// TIA Portal V18 export
TYPE "PLCtoMES_MainCheckOut"
// stored: IsFailsafeCompliant false
   STRUCT
      "P-DataSaveReq" : Bool;   // PLC请求采集质量数据标志位（质量数据全部刷新后触发）MES置位M-DataDone采集完成标志位后，由PLC复位此信号。
      "P-PartType" : String[28];   // PLC请求MES保存时发送产品型号（有RFID则从RFID读取，无RFID，从扫码枪获取）
      "P-PartID" : Array[1..10] of String[48];   // PLC请求MES保存时发送产品序列号（有RFID则从RFID读取，无RFID，从扫码枪获取）
      "P-SubPartID" : Array[1..10] of String[48];   // PLC请求MES保存时发送产品子零件号
      "P-PartResult" : Byte;   // 0-未作，1-合格，2-不合格
      "P-RecipeVer" : String[18];   // 工艺参数版本号
      Reserve : Array[1..1146] of Byte;   // 交互预留
   END_STRUCT;
END_TYPE
